// TIA Portal project "Aufgabe_1_003_mCopilot" (V20)
// *** This TIA Portal project underwent AI modifications via the Siemens Engineering Copilot. ***

(* hardware
DEVICE "S7-1500/ET200MP-Station_1"  S7-1500 station
   slot 0: "Profilschiene_0"  Rack  6ES7 590-1***0-0AA0
   slot 1: "PLC_1"  CPU 1512C-1 PN  6ES7 512-1CK01-0AB0  V2.9
      slot 3: "CPU-Display_1"  6ES7591-1AA00-0AA0
      slot 32768: "PROFINET-Schnittstelle_1"  X1
         slot 32769: "Port_1"  X1 P1
         slot 32770: "Port_2"  X1 P2
      slot 34817: "Virtual CP interface port_1"  Virtual CP interface port  Virtual CP interface port
*)

// ===== PLC "PLC_1"  CPU 1512C-1 PN =====

VAR_GLOBAL   // PLC tag table "Standard-Variablentabelle"
   "x_Start_Prozess" AT %M0.0 : Bool;
   "x_Abgeschlossen" AT %M0.1 : Bool;
END_VAR

VAR_GLOBAL   // PLC tag table "Stanzmaschine"
   "x_Lichtschranke_Ein_Auslagerung" AT %I0.0 : Bool;   // 0 = Werkstueck vorhanden (Oeffner)
   "x_Lichtschranke_Stanzposition" AT %I0.1 : Bool;   // 0 = Werkstueck vorhanden (Oeffner)
   "x_Endlage_Stanze_oben" AT %I0.2 : Bool;   // 1 = Stanze oben (Schliesser)
   "x_Endlage_Stanze_unten" AT %I0.3 : Bool;   // 1 = Stanze oben (Schliesser)
   "x_Motor_Transportband_Vorwaerts" AT %Q0.0 : Bool;   // 1 = Motor laeuft
   "x_Motor_Transportband_Rueckwaerts" AT %Q0.1 : Bool;   // 1 = Motor laeuft
   "x_Motor_Stanze_nach_oben" AT %Q0.2 : Bool;   // 1 = Stanze faehrt aufwaerts
   "x_Motor_Stanze_nach_unten" AT %Q0.3 : Bool;   // 1 = Stanze faehrt abwaerts
END_VAR

TYPE "ST_Werkzeug"
   STRUCT
      i_Werkzeug_ID : Int;
      i_Haltezeit_ms : Int;
      x_Aktiv : Bool;
   END_STRUCT;
END_TYPE

TYPE "ST_Stanzprozess"
   STRUCT
      x_Ausfuehren : Bool;
      x_Fertig : Bool;
      x_Stanze_hoch : Bool;
      x_Stanze_runter : Bool;
   END_STRUCT;
END_TYPE

TYPE "LogEntry"
   STRUCT
      Zeitstempel : DTL;
      Schritt : Int;
   END_STRUCT;
END_TYPE

DATA_BLOCK "FB_Werkstuecktransport_DB"   // DB1
{ S7_Optimized_Access := 'TRUE' }
VERSION : 0.1
// stored: InstanceOfName FB_Werkstuecktransport
"FB_Werkstuecktransport"
BEGIN
END_DATA_BLOCK

DATA_BLOCK "Test_DB"   // DB2
{ S7_Optimized_Access := 'TRUE' }
VERSION : 0.1
   VAR
      i_Schritt : Int;
   END_VAR
BEGIN
END_DATA_BLOCK

DATA_BLOCK "DB_Log"   // DB3
{ S7_Optimized_Access := 'TRUE' }
VERSION : 0.1
   VAR
      Eintrag : Array[0..99] of "LogEntry";
   END_VAR
BEGIN
END_DATA_BLOCK

FUNCTION_BLOCK "FB_Stanzprozess"   // FB11, SCL
{ S7_Optimized_Access := 'TRUE' }
VERSION : 0.1
   VAR_INPUT
      x_Ausfuehren : Bool;
      x_Stanze_oben : Bool;
      x_Stanze_unten : Bool;
   END_VAR
   VAR_OUTPUT
      x_Fertig : Bool;
      x_Stanze_hoch : Bool;
      x_Stanze_runter : Bool;
   END_VAR
   VAR
      x_Prozess_aktiv : Bool;
      x_Abwaerts_fertig : Bool;
      x_Haltezeit_aktiv : Bool;
      x_Aufwaerts_fertig : Bool;
      x_Ausfuehren_alt : Bool;
      x_Flanke : Bool;
      time_TON_Haltezeit : TON_TIME;
   END_VAR
BEGIN
   REGION INFO HEADER
       //===============================================================================
       //-------------------------------------------------------------------------------
       // Title:            FB_Stanzprozess
       // Comment/Function: Mit diesem Funktionsbaustein wird der Stanzprozess durchgeführt. Dieser Mechanismus
       //                   führt den eigentlichen Bearbeitungsvorgang am Werkstück durch. Er wird von zwei Motoren
       //                   angetrieben. Ein Motor Stanze aufwärts hebt den Stanzstempel, und ein Motor Stanze
       //                   abwärts senkt ihn zum Stanzen. Die Position des Stanzstempels wird durch zwei
       //                   Endlagen-Sensoren überwacht. Eine Endlage Stanze oben signalisiert, wenn der Stempel
       //                   vollständig angehoben ist, und eine Endlage Stanze unten zeigt an, wenn der Stempel
       //                   die unterste Position erreicht hat.
       // Library/Family:   N.A
       // Author:           ---
       // Tested with:      S7-1500 CPU 1512C-1 PN DC/DC/DC FW 2.9
       // Engineering:      TIA Portal V20
       // Requirements:     --- 
       //-------------------------------------------------------------------------------
       // Change log table:
       // Version  | Date       | Expert in charge        | Changes applied
       //----------|------------|-------------------------|-----------------------------
       // 01.00.00 | 10.12.2025 |          N.N            | First released version
       //===============================================================================
   END_REGION INFO HEADER

   REGION PROCESS
       #x_Flanke := #x_Ausfuehren AND NOT #x_Ausfuehren_alt;
       #x_Ausfuehren_alt := #x_Ausfuehren;

       IF #x_Flanke AND NOT #x_Prozess_aktiv THEN
           #x_Prozess_aktiv := TRUE;
           #x_Fertig := FALSE;
           #x_Abwaerts_fertig := FALSE;
           #x_Haltezeit_aktiv := FALSE;
           #x_Aufwaerts_fertig := FALSE;
       END_IF;

       IF #x_Prozess_aktiv THEN

           IF NOT #x_Abwaerts_fertig THEN
               #x_Stanze_runter := TRUE;
               #x_Stanze_hoch := FALSE;

               IF #x_Stanze_unten THEN
                   #x_Stanze_runter := FALSE;
                   #x_Abwaerts_fertig := TRUE;
                   #x_Haltezeit_aktiv := TRUE;
               END_IF;
           END_IF;

           #time_TON_Haltezeit(IN := #x_Haltezeit_aktiv,
                               PT := T#500ms);

           IF #time_TON_Haltezeit.Q AND #x_Haltezeit_aktiv THEN
               #x_Haltezeit_aktiv := FALSE;
           END_IF;

           IF #x_Abwaerts_fertig AND NOT #x_Haltezeit_aktiv AND NOT #x_Aufwaerts_fertig THEN
               #x_Stanze_hoch := TRUE;
               #x_Stanze_runter := FALSE;

               IF #x_Stanze_oben THEN
                   #x_Stanze_hoch := FALSE;
                   #x_Aufwaerts_fertig := TRUE;
               END_IF;
           END_IF;

           IF #x_Aufwaerts_fertig THEN
               #x_Fertig := TRUE;
               #x_Prozess_aktiv := FALSE;
           END_IF;

       ELSE
           #x_Stanze_hoch := FALSE;
           #x_Stanze_runter := FALSE;
       END_IF;

       IF #x_Stanze_hoch AND #x_Stanze_runter THEN
           #x_Stanze_hoch := FALSE;
           #x_Stanze_runter := FALSE;
       END_IF;

   END_REGION PROCESS
END_FUNCTION_BLOCK

FUNCTION_BLOCK "FB_Werkstuecktransport"   // FB13, SCL
{ S7_Optimized_Access := 'TRUE' }
VERSION : 0.1
   VAR_INPUT
      x_StanzeOben : Bool;
      x_StanzeUnten : Bool;
      x_EinAuslagerung : Bool;
      x_Stanzposition : Bool;
   END_VAR
   VAR_OUTPUT
      x_Transportband_vorwaerts : Bool;
      x_Transportband_rueckwaerts : Bool;
      x_StanzeHoch : Bool;
      x_StanzeRunter : Bool;
      i_AktuellerSchritt : Int := 0;
   END_VAR
BEGIN
END_FUNCTION_BLOCK

FUNCTION "FC_Check" : Void   // FC1, SCL
{ S7_Optimized_Access := 'TRUE' }
VERSION : 0.1
BEGIN
   //Funktionsinhalt nur zur Ueberpruefung der korrekten Verknuepfung des Projekts,
   //mit dem Engineering Copilot
   //
   //Rechenaufgabe
   //Berechne den Quotienten von 32 und 2
END_FUNCTION

FUNCTION "FC_Log" : Void   // FC4, SCL
{ S7_Optimized_Access := 'TRUE' }
VERSION : 0.1
   VAR_INPUT
      i_Schritt : Int;
      dtl_Systemzeit : DTL;
   END_VAR
   VAR_IN_OUT
      i_naechsterEintrag : Int;
   END_VAR
BEGIN
   REGION INFO HEADER
       //===============================================================================
       //-------------------------------------------------------------------------------
       // Title:            FC_Log
       // Comment/Function: Diese Funktion dient zur Protokollierung von Schrittwechseln einer Schrittkette.
       //                   Sie nimmt eine Schrittnummer und einen Zeitstempel entgegen und schreibt
       //                   diese in einen globalen Datenbaustein ("DB_Log"), der als Ringpuffer
       //                   konfiguriert ist.
       // Library/Family:   N.A
       // Author:           ---
       // Tested with:      S7-1500 CPU 1512C-1 PN DC/DC/DC FW 2.9
       // Engineering:      TIA Portal V20
       // Requirements:     --- 
       //-------------------------------------------------------------------------------
       // Change log table:
       // Version  | Date       | Expert in charge        | Changes applied
       //----------|------------|-------------------------|-----------------------------
       // 01.00.00 | 10.12.2025 |          N.N            | First released version
       //===============================================================================
   END_REGION INFO HEADER

   REGION LOG
   // Schritt 1: Die übergebenen Daten (Zeitstempel und Schrittnummer) werden in das
   // Array "Entries" im "DB_Log" geschrieben. Die Position im Array wird durch
   // die Variable "Index" aus demselben DB bestimmt.
       "DB_Log".Eintrag[#i_naechsterEintrag].Zeitstempel := #dtl_Systemzeit;
       "DB_Log".Eintrag[#i_naechsterEintrag].Schritt := #i_Schritt;

   // Schritt 2: Der Index wird um 1 erhöht, um auf die nächste freie Position
   // im Array für den nächsten Schreibvorgang zu zeigen.
   #i_naechsterEintrag := #i_naechsterEintrag + 1;

   // Schritt 3: Es wird geprüft, ob der Index das Ende des Arrays (hier: 100)
   // erreicht hat. Falls ja, wird er auf 0 zurückgesetzt. Dieses Verhalten
   // nennt man Ringpuffer: Wenn das Ende erreicht ist, wird der älteste
   // Eintrag überschrieben.
   IF #i_naechsterEintrag >= 100 THEN
       #i_naechsterEintrag := 0; // Index auf Anfang zurücksetzen
   END_IF;

   END_REGION LOG
END_FUNCTION

ORGANIZATION_BLOCK "Main"   // OB1, FBD, ProgramCycle
TITLE = "Main Program Sweep (Cycle)"
{ S7_Optimized_Access := 'TRUE' }
VERSION : 0.1
   VAR_INPUT
      Initial_Call : Bool;   // Initial call of this OB
      Remanence : Bool;   // =True, if remanent data are available
   END_VAR
BEGIN

REGION Network 1: FB_Werkstuecktransport
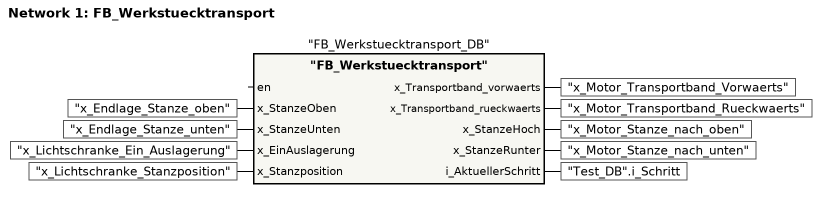
   "FB_Werkstuecktransport_DB"(x_StanzeOben := "x_Endlage_Stanze_oben",   // "FB_Werkstuecktransport"
                           x_StanzeUnten := "x_Endlage_Stanze_unten",
                           x_EinAuslagerung := "x_Lichtschranke_Ein_Auslagerung",
                           x_Stanzposition := "x_Lichtschranke_Stanzposition",
                           x_Transportband_vorwaerts => "x_Motor_Transportband_Vorwaerts",
                           x_Transportband_rueckwaerts => "x_Motor_Transportband_Rueckwaerts",
                           x_StanzeHoch => "x_Motor_Stanze_nach_oben",
                           x_StanzeRunter => "x_Motor_Stanze_nach_unten",
                           i_AktuellerSchritt => "Test_DB".i_Schritt);
END_REGION
END_ORGANIZATION_BLOCK